Staubli VAL3: GenericConv.dtx

bool bClockEnabled
bool bEnableQueuing = true
bool bInit
public bool bLinear = true
bool bLockQueueAcces
public bool bLog
bool bResetConv
public bool bUseUserCenter
public bool bUseUserLimit
dio doClock
public frame fConveyor = {fatherId=world[0]}
public frame fDetection = {fatherId=world[0]}
num nA1 = 1
num nA2 = 1
num nAddedToQueue
num nB1 = 1
num nB2 = 1
num nBoundaryDwn
num nBoundaryUp
public num nBufferSize = 10
public num nCalibratedDist
num nCalibratedID = -99
public num nClockPeriod
public num nConveyorSpeed
num nDEFAULTID = -99
num nDETECT_OVR
public num nDetection2Rob
public num nENCRESOLUTION = 1024
public num nENCSCALEFACTOR
num nEncLatchedVal
num nErrVal[4]
public num nFirDelay
public num nFirOrdre = 20
num nFirTime
num nIdxCalib
num nIdxPull
num nIdxPush
public num nLatchLockDist
num nNumbOfUser
num nPUSH_NEGATIVE
public num nPosMatchTol = 5
num nQueueID = -1
num nStatus = -1
num nSysCycleTime = 0.004
num nTmpEncLatched
num nTmpID
public num nTrackWinHeight = 500
num nWinDownStream
num nWinUpStream
pointRs pObjectRS = {fatherId=world[0]}
pointRx pObject = {fatherId=world[0]}
public string sClockSigName = "none"
string sConvNum
public string sConveyorName = "GenericConv"
public string sDetectionLib = "GenericDetect"
public string sDwnLimSigName = "none"
public string sEncoderLib = "GenericEnc"
string sErrMsgList[12]
  [0] = "Success"
  [1] = "No object available (ID=*)"
  [3] = "The encoder library is not started yet."
  [4] = "The detection library is not started yet."
  [6] = "Run-time error from Conveyor library in task called *\../*. Error code is *"
  [7] = "Run-time error from Encoder library. Error code is *"
  [8] = "Run-time error from Detection library. Error code is *"
  [10] = "Warning, object with negative ID cannot be pushed into conveyor's queue"
  [11] = "Warning, detection overrun."
string sErrorMessage
public string sGeometryLib = "Geometry"
string sMsg
string sTASK[3]
  [0] = "conveyor"
  [1] = "encoder"
  [2] = "detect"
public string sUpLimSigName = "none"
trsf trBoundaryDwn[2]
trsf trBoundaryUp[2]
trsf trDEFAULT = {x=5, y=4, z=3, rx=2, ry=1}
trsf trDetectedCoord
trsf trTmp
